// TIA Portal V20 export
FUNCTION_BLOCK "FB_LightsManagement"   // FB500, SCL
{ S7_Optimized_Access := 'TRUE' }
// stored: AutoNumber false, MemoryReserve 100, SetENOAutomatically false
BEGIN
   REGION Light Tower : Green light
       "DB_DigitalOutputs".sLightTowerGreen.sSWStatus :=
       "LBP_Chan1".E_ProgRunning
       OR "LBP_Chan1".E_ProgWait
       OR "LBP_Chan1".E_ProgStop
       OR "DB_McpKeyboardSignals".sLightTest.sKeySWStatus;
   END_REGION

   REGION Light Tower : Orange light
       "DB_DigitalOutputs".sLightTowerOrange.sSWStatus := ("DB_DataFromSafety".iEmergencyStopPowerLaser
       AND "DB_DataFromSafety".ShutterOpened
       AND "Clock_2.5Hz")
       OR "DB_McpKeyboardSignals".sLightTest.sKeySWStatus;
   END_REGION

   REGION Light Tower : Blue light
       "DB_DigitalOutputs".sLightTowerBlue.sSWStatus :=
       ("LBP_ModeGroup".E_AUTO
       AND ("LBP_Chan1".E_ProgRunning OR "LBP_Chan1".E_ProgWait)
       AND NOT "DB_DataFromSafety".EmergencyStop    
       AND "Clock_1Hz")
       OR "DB_McpKeyboardSignals".sLightTest.sKeySWStatus;
   END_REGION

   REGION Light Tower : White light
       "DB_DigitalOutputs".sLightTowerWhite.sSWStatus :=
       ("DB_PowerOn".sMachinePower
       AND "Clock_0.625Hz")
       OR "DB_McpKeyboardSignals".sLightTest.sKeySWStatus;
   END_REGION

   REGION Test LED light
       "DB_McpKeyboardSignals".sLightTest.sLedSWStatus := "DB_McpKeyboardSignals".sLightTest.sKeySWStatus;
   END_REGION

   REGION Machine lights (Key K15)
       IF "DB_McpKeyboardSignals".sK15_MachineLight.sKeySWTogglePositiveFront
           OR "DB_HmiKeyboardSignals".sK15_MachineLight.sKeySWTogglePositiveFront THEN
           "DB_DigitalOutputs".sMachineLight.sSWStatus := TRUE;
           "DB_DigitalOutputs".sMachineLightBack.sSWStatus := TRUE;
           "DB_McpKeyboardSignals".sK15_MachineLight.sKeySWToggleStatus := TRUE;
           "DB_HmiKeyboardSignals".sK15_MachineLight.sKeySWToggleStatus := TRUE;
       ELSIF "DB_McpKeyboardSignals".sK15_MachineLight.sKeySWToggleNegativeFront
           OR "DB_HmiKeyboardSignals".sK15_MachineLight.sKeySWToggleNegativeFront THEN
           "DB_DigitalOutputs".sMachineLight.sSWStatus := FALSE;
           "DB_DigitalOutputs".sMachineLightBack.sSWStatus := FALSE;
           "DB_McpKeyboardSignals".sK15_MachineLight.sKeySWToggleStatus := FALSE;
           "DB_HmiKeyboardSignals".sK15_MachineLight.sKeySWToggleStatus := FALSE;
       END_IF;
           "DB_McpKeyboardSignals".sK15_MachineLight.sLedSWStatus := "DB_DigitalOutputs".sMachineLight.sSWStatus;
           "DB_HmiKeyboardSignals".sK15_MachineLight.sLedSWStatus := "DB_DigitalOutputs".sMachineLight.sSWStatus;
   END_REGION

   REGION Camera lights (Key K12)    
       IF "LBP_Chan1".MDyn[50] THEN
           "DB_McpKeyboardSignals".sK12_ObservationCamera.sKeySWToggleStatus := TRUE;
           "DB_HmiKeyboardSignals".sK12b_ObservationCamera.sKeySWToggleStatus := TRUE;
       ELSIF "LBP_Chan1".MDyn[51] THEN
           "DB_McpKeyboardSignals".sK12_ObservationCamera.sKeySWToggleStatus := FALSE;
           "DB_HmiKeyboardSignals".sK12b_ObservationCamera.sKeySWToggleStatus := FALSE;
       END_IF;

       IF "DB_McpKeyboardSignals".sK12_ObservationCamera.sKeySWTogglePositiveFront
           OR "DB_HmiKeyboardSignals".sK12a_Backlight.sKeySWTogglePositiveFront THEN
           "DB_DigitalOutputs".sBacklight.sSWStatus := TRUE;
       ELSIF "DB_McpKeyboardSignals".sK12_ObservationCamera.sKeySWToggleNegativeFront
           OR "DB_HmiKeyboardSignals".sK12a_Backlight.sKeySWToggleNegativeFront THEN
           "DB_DigitalOutputs".sBacklight.sSWStatus := FALSE;
       END_IF;

       "DB_McpKeyboardSignals".sK12_ObservationCamera.sLedSWStatus := "DB_DigitalOutputs".sBacklight.sSWStatus;
       "DB_HmiKeyboardSignals".sK12a_Backlight.sLedSWStatus := "DB_DigitalOutputs".sBacklight.sSWStatus;

       IF "DB_McpKeyboardSignals".sK12_ObservationCamera.sKeySWTogglePositiveFront
           OR "DB_HmiKeyboardSignals".sK12b_ObservationCamera.sKeySWTogglePositiveFront THEN
           "DB_DigitalOutputs".sObservationCameraLight.sSWStatus := TRUE;
       ELSIF "DB_McpKeyboardSignals".sK12_ObservationCamera.sKeySWToggleNegativeFront
           OR "DB_HmiKeyboardSignals".sK12b_ObservationCamera.sKeySWToggleNegativeFront THEN
           "DB_DigitalOutputs".sObservationCameraLight.sSWStatus := FALSE;
       END_IF;

       "DB_McpKeyboardSignals".sK12_ObservationCamera.sLedSWStatus := "DB_DigitalOutputs".sObservationCameraLight.sSWStatus;
       "DB_HmiKeyboardSignals".sK12b_ObservationCamera.sLedSWStatus := "DB_DigitalOutputs".sObservationCameraLight.sSWStatus;
   END_REGION

   REGION Ack blue button AND red light tower blinking
       "DB_McpKeyboardSignals".sAlarmReset.sLedSWStatus :=
           (( "DB_Alarms".sAlarmsLevel1
           OR "DB_Alarms".sAlarmsLevel2
           OR "DB_Alarms".sAlarmsLevel3
           OR "DB_Alarms".sAlarmsLevel4
           OR "DB_Alarms".sAlarmsLevel5
           OR "DB_Alarms".sAlarmsLevel6)
           AND "Clock_1Hz")
           OR "DB_McpKeyboardSignals".sLightTest.sKeySWStatus;

           "DB_DigitalOutputs".sLightTowerRed.sSWStatus :=
           (( "DB_Alarms".sAlarmsLevel2
           OR "DB_Alarms".sAlarmsLevel3
           OR "DB_Alarms".sAlarmsLevel4
           OR "DB_Alarms".sAlarmsLevel5
           OR "DB_Alarms".sAlarmsLevel6)
           AND "Clock_1Hz")
           OR "DB_McpKeyboardSignals".sLightTest.sKeySWStatus;
   END_REGION
END_FUNCTION_BLOCK
